FUNCTION_BLOCK FB_Module01 EXTENDS FB_Module
VAR_INPUT
END_VAR
VAR_OUTPUT
END_VAR
VAR
	fbComponent1:				FB_Component;
	fbComponent2:				FB_Component;
	fbComponent3:				FB_Component;
	fbComponent4:				FB_ComponentEX;
END_VAR

METHOD PUBLIC M_Cycle
VAR_INPUT
END_VAR
SUPER^.M_Cycle();

fbComponent1.M_Cycle();
fbComponent2.M_Cycle();
fbComponent3.M_Cycle();
fbComponent4.M_Cycle();
END_METHOD

METHOD PROTECTED M_Initialise : BOOL
VAR_INPUT
END_VAR
M_Initialise:= SUPER^.M_Initialise();

M_Attach(fbComponent1);
M_Attach(fbComponent2);
M_Attach(fbComponent3);
M_Attach(fbComponent4);
END_METHOD

METHOD PROTECTED M_Running
VAR_INPUT
END_VAR
IF NOT M001.fbPowerOn.P_Value THEN
	fbEvent.M_Add(M001.fbPowerOn.P_ID);
	fbEvent.M_Error('Power not on', 2 ,E_Behaviour.Abort);
ELSIF NOT M001.fbFuse1.P_Value THEN
	fbEvent.M_Add(M001.fbFuse1.P_ID);
	fbEvent.M_Error('Fuse Triped', 3 ,E_Behaviour.Stop);	
	
END_IF

fbEvent.M_Warning('My first Warning', 4 );
END_METHOD

END_FUNCTION_BLOCK

(* stored: Version 1.1.0.1, ProductVersion 3.1.4024.12
   POU FB_Module01: Id {3744d03d-359c-4ab8-84fb-4ea93b7a5162}, SpecialFunc None
   Method M_Cycle: Id {655447dc-389e-494a-be91-78d8a111b7aa}
   Method M_Initialise: Id {714c485c-83a6-4af2-a706-fec3f6b598e5}
   Method M_Running: Id {eaffebca-5ff2-4f17-be84-3310a9ace22e} *)
